(* Logix 5000 project; controller Lab7_1 5069-L306ERM rev 35.16; software revision 35.00 *)

TASK MainTask (continuous, watchdog 500 ms) : MainProgram

MODULES
   Local : 5069-L306ERM (5069 0, rev 35.16)
      IOHub : vendor 1 type 7 code 358 (Ethernet 192.168.110.5, rev 1.1, Output RPI 20 ms)
END_MODULES

PROGRAM MainProgram   (* main routine MainRoutine *)
VAR
   displayTimer : TIMER := (PRE := 500);
   Dummy : BOOL;
END_VAR

ROUTINE MainRoutine   (* ladder *)
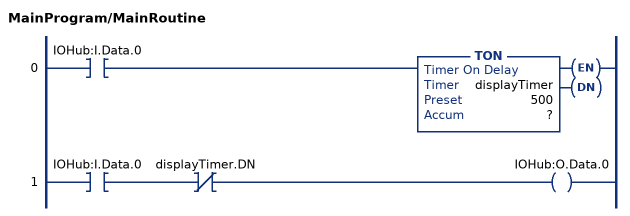
   0: XIC(IOHub:I.Data.0)TON(displayTimer,?,?);
   1: XIC(IOHub:I.Data.0)XIO(displayTimer.DN)OTE(IOHub:O.Data.0);
END_ROUTINE
END_PROGRAM
